FUNCTION TemplateFunction (* Function with empty body *)
  (* Standard: 61499-1 *)
  (* Version 1.0, 2023-06-29, mjobst, 4DIAC-Consortium *)
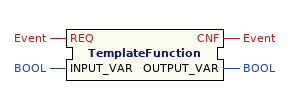
  EVENT_INPUT
    REQ;
  END_EVENT
  EVENT_OUTPUT
    CNF;
  END_EVENT
  VAR_INPUT
    INPUT_VAR : BOOL; (* Input variable *)
  END_VAR
  VAR_OUTPUT
    OUTPUT_VAR : BOOL; (* Output variable (normally not used!) *)
  END_VAR
END_FUNCTION
